KUKA KRL program: wkz6_an.src, wkz6_an.dat

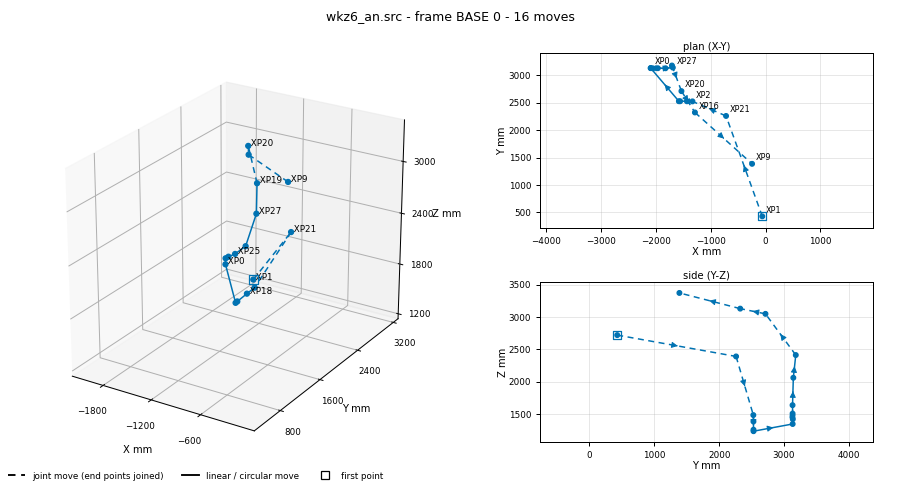
[picture p0: tool path of wkz6_an.src in frame BASE 0, 16 of 16 moves have a stored position in this frame; points joined in program order, loops and branches not executed]
--- wkz6_an.src ---
&ACCESS RVO4
&REL 71
&COMMENT Peg Grp AXOR
&PARAM DISKPATH = KRC:\R1\Program
&PARAM TEMPLATE = C:\KRC\Roboter\Template\vorgabe
&PARAM EDITMASK = *
DEF wkz6_an( )
;FOLD INI
  ;FOLD BASISTECH INI
    GLOBAL INTERRUPT DECL 3 WHEN $STOPMESS==TRUE DO IR_STOPM ( )
    INTERRUPT ON 3
    BAS (#INITMOV,0 )
  ;ENDFOLD (BASISTECH INI)
;FOLD GRIPPERTECH INI
USER_GRP(0,DUMMY,DUMMY,GDEFAULT)
;ENDFOLD (GRIPPERTECH INI)
  ;FOLD USER INI
    ;Make your modifications here

  ;ENDFOLD (USER INI)
;ENDFOLD (INI)

; Caracterização dos meios de produção
; Changes: Pega Gripper Axor/Atego
; Versão Atual:02/08/2015
; Name: P13.050-R3
; Docking

chk_w8_wechs_ok ( )     ; CHECK TOOL CHANGE

;FOLD PTP P1 CONT Vel=100 % PDAT1 Tool[6]:Gripper G0100R Base[0];%{PE}%R 8.2.20,%MKUKATPBASIS,%CMOVE,%VPTP,%P 1:PTP, 2:P1, 3:C_DIS, 5:100, 7:PDAT1
$BWDSTART=FALSE
PDAT_ACT=PPDAT1
FDAT_ACT=FP1
BAS(#PTP_PARAMS,100)
PTP XP1 C_DIS
;ENDFOLD

;FOLD WAIT FOR NOT ( IN 219 'Posicao p/ Acoplamento OK' ) CONT;%{PE}%R 8.2.20,%MKUKATPBASIS,%CEXT_WAIT_FOR,%VEXT_WAIT_FOR,%P 2:NOT, 4:, 5:$IN, 6:219, 7:Posicao p/ Acoplamento OK, 9:CONTINUE
CONTINUE
WAIT FOR  NOT ( $IN[219] )
;ENDFOLD
;FOLD WAIT FOR ( IN 201 'DOCK 6 Deposito Ocupado' ) CONT;%{PE}%R 8.2.20,%MKUKATPBASIS,%CEXT_WAIT_FOR,%VEXT_WAIT_FOR,%P 2:, 4:, 5:$IN, 6:201, 7:DOCK 6 Deposito Ocupado, 9:CONTINUE
CONTINUE
WAIT FOR  ( $IN[201] )
;ENDFOLD
;FOLD PULSE 207 'DOCK 6 Abrir Proteção' State=TRUE CONT Time=1 sec;%{PE}%R 8.2.20,%MKUKATPBASIS,%COUT,%VPULSE,%P 2:207, 3:DOCK 6 Abrir Proteção, 5:TRUE, 6:CONTINUE, 8:1
CONTINUE
PULSE($OUT[207], TRUE,1)
;ENDFOLD

;FOLD PTP P21 CONT Vel=100 % PDAT16 Tool[6]:Gripper G0100R Base[0];%{PE}%R 8.2.20,%MKUKATPBASIS,%CMOVE,%VPTP,%P 1:PTP, 2:P21, 3:C_DIS, 5:100, 7:PDAT16
$BWDSTART=FALSE
PDAT_ACT=PPDAT16
FDAT_ACT=FP21
BAS(#PTP_PARAMS,100)
PTP XP21 C_DIS
;ENDFOLD

;FOLD WAIT FOR ( IN 205 'DOCK 6 Proteção Aberta' ) CONT;%{PE}%R 8.2.20,%MKUKATPBASIS,%CEXT_WAIT_FOR,%VEXT_WAIT_FOR,%P 2:, 4:, 5:$IN, 6:205, 7:DOCK 6 Proteção Aberta, 9:CONTINUE
CONTINUE
WAIT FOR  ( $IN[205] )
;ENDFOLD
;FOLD WAIT FOR NOT ( IN 206 'DOCK 6 Proteção Fechada' ) CONT;%{PE}%R 8.2.20,%MKUKATPBASIS,%CEXT_WAIT_FOR,%VEXT_WAIT_FOR,%P 2:NOT, 4:, 5:$IN, 6:206, 7:DOCK 6 Proteção Fechada, 9:CONTINUE
CONTINUE
WAIT FOR  NOT ( $IN[206] )
;ENDFOLD

;FOLD PTP P2 CONT Vel=100 % PDAT7 Tool[6]:Gripper G0100R Base[0];%{PE}%R 8.2.20,%MKUKATPBASIS,%CMOVE,%VPTP,%P 1:PTP, 2:P2, 3:C_DIS, 5:100, 7:PDAT7
$BWDSTART=FALSE
PDAT_ACT=PPDAT7
FDAT_ACT=FP2
BAS(#PTP_PARAMS,100)
PTP XP2 C_DIS
;ENDFOLD
;FOLD LIN P18 CONT Vel=1 m/s CPDAT9 Tool[6]:Gripper G0100R Base[0];%{PE}%R 8.2.20,%MKUKATPBASIS,%CMOVE,%VLIN,%P 1:LIN, 2:P18, 3:C_DIS C_DIS, 5:1, 7:CPDAT9
$BWDSTART=FALSE
LDAT_ACT=LCPDAT9
FDAT_ACT=FP18
BAS(#CP_PARAMS,1)
LIN XP18 C_DIS C_DIS
;ENDFOLD
;FOLD LIN P22 CONT Vel=1 m/s CPDAT0 Tool[6]:Gripper G0100R Base[0];%{PE}%R 8.2.20,%MKUKATPBASIS,%CMOVE,%VLIN,%P 1:LIN, 2:P22, 3:C_DIS C_DIS, 5:1, 7:CPDAT0
$BWDSTART=FALSE
LDAT_ACT=LCPDAT0
FDAT_ACT=FP22
BAS(#CP_PARAMS,1)
LIN XP22 C_DIS C_DIS
;ENDFOLD

;FOLD WAIT FOR ( IN 222 'Liberacao p/ Desbloqueio' );%{PE}%R 8.2.20,%MKUKATPBASIS,%CEXT_WAIT_FOR,%VEXT_WAIT_FOR,%P 2:, 4:, 5:$IN, 6:222, 7:Liberacao p/ Desbloqueio, 9:
WAIT FOR  ( $IN[222] )
;ENDFOLD
;FOLD OUT 224 'Bloquear MPS' State=FALSE ;%{PE}%R 8.2.20,%MKUKATPBASIS,%COUT,%VOUTX,%P 2:224, 3:Bloquear MPS, 5:FALSE, 6:
$OUT[224]=FALSE
;ENDFOLD
;FOLD OUT 223 'Desbloquear MPS' State=TRUE ;%{PE}%R 8.2.20,%MKUKATPBASIS,%COUT,%VOUTX,%P 2:223, 3:Desbloquear MPS, 5:TRUE, 6:
$OUT[223]=TRUE
;ENDFOLD
;FOLD WAIT FOR ( IN 217 'MPS Destravado' );%{PE}%R 8.2.20,%MKUKATPBASIS,%CEXT_WAIT_FOR,%VEXT_WAIT_FOR,%P 2:, 4:, 5:$IN, 6:217, 7:MPS Destravado, 9:
WAIT FOR  ( $IN[217] )
;ENDFOLD
;FOLD WAIT FOR NOT ( IN 221 'MPS Travado' );%{PE}%R 8.2.20,%MKUKATPBASIS,%CEXT_WAIT_FOR,%VEXT_WAIT_FOR,%P 2:NOT, 4:, 5:$IN, 6:221, 7:MPS Travado, 9:
WAIT FOR  NOT ( $IN[221] )
;ENDFOLD

;FOLD ; POSICAO DE PEGA DO GRIPPER NO DOCKING;%{PE}%R 8.2.17,%MKUKATPBASIS,%CCOMMENT,%VNORMAL,%P 2:POSICAO DE PEGA DO GRIPPER NO DOCKING
;ENDFOLD
;FOLD LIN P4 Vel=0.2 m/s CPDAT16 Tool[8]:Tool Changer Base[0];%{PE}%R 8.2.20,%MKUKATPBASIS,%CMOVE,%VLIN,%P 1:LIN, 2:P4, 3:, 5:0.2, 7:CPDAT16
$BWDSTART=FALSE
LDAT_ACT=LCPDAT16
FDAT_ACT=FP4
BAS(#CP_PARAMS,0.2)
LIN XP4
;ENDFOLD

;FOLD WAIT FOR ( IN 219 'Posicao p/ Acoplamento OK' );%{PE}%R 8.2.20,%MKUKATPBASIS,%CEXT_WAIT_FOR,%VEXT_WAIT_FOR,%P 2:, 4:, 5:$IN, 6:219, 7:Posicao p/ Acoplamento OK, 9:
WAIT FOR  ( $IN[219] )
;ENDFOLD
;FOLD WAIT Time=0.5 sec;%{PE}%R 8.2.20,%MKUKATPBASIS,%CWAIT,%VWAIT,%P 3:0.5
WAIT SEC 0.5
;ENDFOLD
;FOLD OUT 223 'Desbloquear MPS' State=FALSE ;%{PE}%R 8.2.20,%MKUKATPBASIS,%COUT,%VOUTX,%P 2:223, 3:Desbloquear MPS, 5:FALSE, 6:
$OUT[223]=FALSE
;ENDFOLD
;FOLD OUT 224 'Bloquear MPS' State=TRUE ;%{PE}%R 8.2.20,%MKUKATPBASIS,%COUT,%VOUTX,%P 2:224, 3:Bloquear MPS, 5:TRUE, 6:
$OUT[224]=TRUE
;ENDFOLD
;FOLD WAIT FOR NOT ( IN 217 'MPS Destravado' );%{PE}%R 8.2.20,%MKUKATPBASIS,%CEXT_WAIT_FOR,%VEXT_WAIT_FOR,%P 2:NOT, 4:, 5:$IN, 6:217, 7:MPS Destravado, 9:
WAIT FOR  NOT ( $IN[217] )
;ENDFOLD
;FOLD WAIT FOR ( IN 221 'MPS Travado' );%{PE}%R 8.2.20,%MKUKATPBASIS,%CEXT_WAIT_FOR,%VEXT_WAIT_FOR,%P 2:, 4:, 5:$IN, 6:221, 7:MPS Travado, 9:
WAIT FOR  ( $IN[221] )
;ENDFOLD
;FOLD IBUS ON SEGMENT_4;%{PE}%R 8.2.20,%MKUKATPBASIS,%CIBUS,%VMAP,%P 2:#ON, 3:4
$IBUS_ON=IBUS_SEGMENT[4]
$IBUS_OFF=0
;ENDFOLD
;FOLD WAIT Time=0.5 sec;%{PE}%R 8.2.20,%MKUKATPBASIS,%CWAIT,%VWAIT,%P 3:0.5
WAIT SEC 0.5
;ENDFOLD

; Verifica Grampos da Garra Fechados
chk_w6_grp3_clo()
chk_w6_grp4_clo()
chk_w6_grp5_clo()
chk_w6_grp6_clo()
chk_w6_grp7_clo()

;FOLD LIN P0 CONT Vel=0.3 m/s CPDAT1 Tool[6]:Gripper G0100R Base[0];%{PE}%R 8.2.20,%MKUKATPBASIS,%CMOVE,%VLIN,%P 1:LIN, 2:P0, 3:C_DIS C_DIS, 5:0.3, 7:CPDAT1
$BWDSTART=FALSE
LDAT_ACT=LCPDAT1
FDAT_ACT=FP0
BAS(#CP_PARAMS,0.3)
LIN XP0 C_DIS C_DIS
;ENDFOLD
;FOLD LIN P12 CONT Vel=0.5 m/s CPDAT7 Tool[6]:Gripper G0100R Base[0];%{PE}%R 8.2.20,%MKUKATPBASIS,%CMOVE,%VLIN,%P 1:LIN, 2:P12, 3:C_DIS C_DIS, 5:0.5, 7:CPDAT7
$BWDSTART=FALSE
LDAT_ACT=LCPDAT7
FDAT_ACT=FP12
BAS(#CP_PARAMS,0.5)
LIN XP12 C_DIS C_DIS
;ENDFOLD

;FOLD WAIT FOR NOT ( IN 201 'DOCK 6 Deposito Ocupado' ) CONT;%{PE}%R 8.2.20,%MKUKATPBASIS,%CEXT_WAIT_FOR,%VEXT_WAIT_FOR,%P 2:NOT, 4:, 5:$IN, 6:201, 7:DOCK 6 Deposito Ocupado, 9:CONTINUE
CONTINUE
WAIT FOR  NOT ( $IN[201] )
;ENDFOLD
;FOLD WAIT FOR ( IN 219 'Posicao p/ Acoplamento OK' ) CONT;%{PE}%R 8.2.20,%MKUKATPBASIS,%CEXT_WAIT_FOR,%VEXT_WAIT_FOR,%P 2:, 4:, 5:$IN, 6:219, 7:Posicao p/ Acoplamento OK, 9:CONTINUE
CONTINUE
WAIT FOR  ( $IN[219] )
;ENDFOLD

;FOLD LIN P24 CONT Vel=1 m/s CPDAT11 Tool[6]:Gripper G0100R Base[0];%{PE}%R 8.2.20,%MKUKATPBASIS,%CMOVE,%VLIN,%P 1:LIN, 2:P24, 3:C_DIS C_DIS, 5:1, 7:CPDAT11
$BWDSTART=FALSE
LDAT_ACT=LCPDAT11
FDAT_ACT=FP24
BAS(#CP_PARAMS,1)
LIN XP24 C_DIS C_DIS
;ENDFOLD
;FOLD LIN P25 CONT Vel=1 m/s CPDAT17 Tool[6]:Gripper G0100R Base[0];%{PE}%R 8.2.20,%MKUKATPBASIS,%CMOVE,%VLIN,%P 1:LIN, 2:P25, 3:C_DIS C_DIS, 5:1, 7:CPDAT17
$BWDSTART=FALSE
LDAT_ACT=LCPDAT17
FDAT_ACT=FP25
BAS(#CP_PARAMS,1)
LIN XP25 C_DIS C_DIS
;ENDFOLD
;FOLD LIN P26 CONT Vel=1 m/s CPDAT18 Tool[6]:Gripper G0100R Base[0];%{PE}%R 8.2.20,%MKUKATPBASIS,%CMOVE,%VLIN,%P 1:LIN, 2:P26, 3:C_DIS C_DIS, 5:1, 7:CPDAT18
$BWDSTART=FALSE
LDAT_ACT=LCPDAT18
FDAT_ACT=FP26
BAS(#CP_PARAMS,1)
LIN XP26 C_DIS C_DIS
;ENDFOLD
;FOLD LIN P27 CONT Vel=2 m/s CPDAT19 Tool[6]:Gripper G0100R Base[0];%{PE}%R 8.2.20,%MKUKATPBASIS,%CMOVE,%VLIN,%P 1:LIN, 2:P27, 3:C_DIS C_DIS, 5:2, 7:CPDAT19
$BWDSTART=FALSE
LDAT_ACT=LCPDAT19
FDAT_ACT=FP27
BAS(#CP_PARAMS,2)
LIN XP27 C_DIS C_DIS
;ENDFOLD
;FOLD LIN P19 CONT Vel=2 m/s CPDAT15 Tool[6]:Gripper G0100R Base[0];%{PE}%R 8.2.20,%MKUKATPBASIS,%CMOVE,%VLIN,%P 1:LIN, 2:P19, 3:C_DIS C_DIS, 5:2, 7:CPDAT15
$BWDSTART=FALSE
LDAT_ACT=LCPDAT15
FDAT_ACT=FP19
BAS(#CP_PARAMS,2)
LIN XP19 C_DIS C_DIS
;ENDFOLD
;FOLD PTP P20 CONT Vel=100 % PDAT15 Tool[6]:Gripper G0100R Base[0];%{PE}%R 8.2.20,%MKUKATPBASIS,%CMOVE,%VPTP,%P 1:PTP, 2:P20, 3:C_DIS, 5:100, 7:PDAT15
$BWDSTART=FALSE
PDAT_ACT=PPDAT15
FDAT_ACT=FP20
BAS(#PTP_PARAMS,100)
PTP XP20 C_DIS
;ENDFOLD
;FOLD PTP P16 CONT Vel=100 % PDAT12 Tool[6]:Gripper G0100R Base[0];%{PE}%R 8.2.20,%MKUKATPBASIS,%CMOVE,%VPTP,%P 1:PTP, 2:P16, 3:C_DIS, 5:100, 7:PDAT12
$BWDSTART=FALSE
PDAT_ACT=PPDAT12
FDAT_ACT=FP16
BAS(#PTP_PARAMS,100)
PTP XP16 C_DIS
;ENDFOLD
;FOLD PTP P9 CONT Vel=100 % PDAT4 Tool[6]:Gripper G0100R Base[0];%{PE}%R 8.2.20,%MKUKATPBASIS,%CMOVE,%VPTP,%P 1:PTP, 2:P9, 3:C_DIS, 5:100, 7:PDAT4
$BWDSTART=FALSE
PDAT_ACT=PPDAT4
FDAT_ACT=FP9
BAS(#PTP_PARAMS,100)
PTP XP9 C_DIS
;ENDFOLD

END

--- wkz6_an.dat ---
&ACCESS RVO4
&REL 71
&COMMENT Peg Grp AXOR
&PARAM DISKPATH = KRC:\R1\Program
&PARAM TEMPLATE = C:\KRC\Roboter\Template\vorgabe
&PARAM EDITMASK = *
DEFDAT  wkz6_an
;FOLD EXTERNAL DECLARATIONS;%{PE}%MKUKATPBASIS,%CEXT,%VCOMMON,%P
;FOLD GRIPPERTECH EXT
EXT  H50 (INT  :IN,INT  :IN,INT  :IN,GRP_TYP  :IN )
;ENDFOLD (GRIPPERTECH EXT)
;FOLD SPOTTECH EXT
EXT  USERSPOT (S_COMMAND  :IN,SPOT_TYPE  :IN )
;ENDFOLD (SPOTTECH EXT)
;FOLD BASISTECH EXT;%{PE}%MKUKATPBASIS,%CEXT,%VEXT,%P
EXT  BAS (BAS_COMMAND  :IN,REAL  :IN )
DECL INT SUCCESS
;ENDFOLD (BASISTECH EXT)
;FOLD USER EXT;%{E}%MKUKATPUSER,%CEXT,%VEXT,%P
;Make your modifications here

;ENDFOLD (USER EXT)
;ENDFOLD (EXTERNAL DECLARATIONS)
DECL BASIS_SUGG_T LAST_BASIS={POINT1[] "P0                      ",POINT2[] "P0                      ",CP_PARAMS[] "CPDAT0                  ",PTP_PARAMS[] "PDAT0                   ",CONT[] "                        ",CP_VEL[] "0.2                     ",PTP_VEL[] "100                     ",SYNC_PARAMS[] "SYNCDAT                 ",SPL_NAME[] "S0                      "}
DECL E6POS XP2={X -1334.70801,Y 2526.76001,Z 1488.44397,A -20.9060402,B 43.2974091,C 166.070602,S 2,T 10,E1 -276.315094,E2 0.0,E3 0.0,E4 0.0,E5 0.0,E6 0.0}
DECL FDAT FP2={TOOL_NO 8,BASE_NO 0,IPO_FRAME #BASE,POINT2[] " ",TQ_STATE FALSE}
DECL E6POS XP4={X -1582.73999,Y 2529.76489,Z 1240.026,A -20.81633,B 42.8571701,C 165.799393,S 2,T 10,E1 -276.288391,E2 0.0,E3 0.0,E4 0.0,E5 0.0,E6 0.0}
DECL FDAT FP4={TOOL_NO 8,BASE_NO 0,IPO_FRAME #BASE,POINT2[] " ",TQ_STATE FALSE}
DECL E6POS XP9={X -246.532501,Y 1387.03601,Z 3371.896,A -169.795593,B 6.91202211,C 129.772507,S 2,T 34,E1 -430.979797,E2 0.0,E3 0.0,E4 0.0,E5 0.0,E6 0.0}
DECL FDAT FP9={TOOL_NO 6,BASE_NO 0,IPO_FRAME #BASE,POINT2[] " ",TQ_STATE FALSE}
DECL PDAT PPDAT4={VEL 100.0,ACC 100.0,APO_DIST 0.0,APO_MODE #CDIS}
DECL E6POS XP12={X -2096.30688,Y 3135.69604,Z 1425.60205,A -0.0780687928,B 45.1058998,C -104.320198,S 2,T 10,E1 -276.26181,E2 0.0,E3 0.0,E4 0.0,E5 0.0,E6 0.0}
DECL FDAT FP12={TOOL_NO 6,BASE_NO 0,IPO_FRAME #BASE,POINT2[] " ",TQ_STATE FALSE}
DECL LDAT LCPDAT7={VEL 2.0,ACC 100.0,APO_DIST 20.0,APO_FAC 50.0,AXIS_VEL 100.0,AXIS_ACC 100.0,ORI_TYP #VAR,CIRC_TYP #BASE,JERK_FAC 50.0,GEAR_JERK 50.0,EXAX_IGN 0}
DECL PDAT PPDAT7={VEL 100.0,ACC 100.0,APO_DIST 50.0,APO_MODE #CDIS}
DECL E6POS XP16={X -1289.547,Y 2324.76294,Z 3130.05688,A -36.2241287,B 48.9362907,C -95.0278778,S 2,T 34,E1 -331.860504,E2 0.0,E3 0.0,E4 0.0,E5 0.0,E6 0.0}
DECL FDAT FP16={TOOL_NO 6,BASE_NO 0,IPO_FRAME #BASE,POINT2[] " ",TQ_STATE FALSE}
DECL PDAT PPDAT12={VEL 100.0,ACC 100.0,APO_DIST 100.0,APO_MODE #CDIS}
DECL E6POS XP18={X -1434.875,Y 2528.70508,Z 1389.41895,A -20.3609009,B 42.94133,C 166.110596,S 2,T 10,E1 -276.315002,E2 0.0,E3 0.0,E4 0.0,E5 0.0,E6 0.0}
DECL FDAT FP18={TOOL_NO 8,BASE_NO 0,IPO_FRAME #BASE,POINT2[] " ",TQ_STATE FALSE}
DECL LDAT LCPDAT9={VEL 2.0,ACC 100.0,APO_DIST 10.0,APO_FAC 50.0,AXIS_VEL 100.0,AXIS_ACC 100.0,ORI_TYP #VAR,CIRC_TYP #BASE,JERK_FAC 50.0,GEAR_JERK 50.0,EXAX_IGN 0}
DECL E6POS XP19={X -1709.26904,Y 3181.41309,Z 2414.36304,A 0.598406494,B 55.2073517,C -102.179604,S 2,T 10,E1 -276.258514,E2 0.0,E3 0.0,E4 0.0,E5 0.0,E6 0.0}
DECL FDAT FP19={TOOL_NO 6,BASE_NO 0,IPO_FRAME #BASE,POINT2[] " ",TQ_STATE FALSE}
DECL E6POS XP20={X -1535.84998,Y 2714.00806,Z 3049.51196,A 15.8610601,B 57.4065895,C -83.8867493,S 2,T 10,E1 -276.258606,E2 0.0,E3 0.0,E4 0.0,E5 0.0,E6 0.0}
DECL FDAT FP20={TOOL_NO 6,BASE_NO 0,IPO_FRAME #BASE,POINT2[] " ",TQ_STATE FALSE}
DECL PDAT PPDAT15={VEL 100.0,ACC 100.0,APO_DIST 100.0,APO_MODE #CDIS}
DECL GRP_SUGG_T LAST_GRP={NUMBER[] "14                      ",STATE[] "2                       ",PARAMS[] "GDAT5                   "}
DECL GRP_TYP GGDAT14={G_APO #NO,GRP_TIME 0.200000003,CTRL #OFF,DLY 0,DST 1}
DECL GRP_TYP GGDAT15={G_APO #NO,GRP_TIME 0.200000003,CTRL #OFF,DLY 0,DST 1}
DECL GRP_TYP GGDAT16={G_APO #NO,GRP_TIME 0.200000003,CTRL #OFF,DLY 0,DST 1}
DECL GRP_TYP GGDAT17={G_APO #NO,GRP_TIME 0.200000003,CTRL #OFF,DLY 0,DST 1}
DECL GRP_TYP GGDAT18={G_APO #NO,GRP_TIME 0.200000003,CTRL #OFF,DLY 0,DST 1}
DECL GRP_TYP GGDAT19={G_APO #NO,GRP_TIME 0.200000003,CTRL #OFF,DLY 0,DST 1}
DECL E6POS XP21={X -721.451416,Y 2260.86401,Z 2392.80103,A -69.6591873,B 42.6547394,C -179.8293,S 2,T 10,E1 -276.320099,E2 0.0,E3 0.0,E4 0.0,E5 0.0,E6 0.0}
DECL FDAT FP21={TOOL_NO 8,BASE_NO 0,IPO_FRAME #BASE,POINT2[] " ",TQ_STATE FALSE}
DECL PDAT PPDAT16={VEL 100.0,ACC 100.0,APO_DIST 100.0,APO_MODE #CDIS}
DECL LDAT LCPDAT0={VEL 2.0,ACC 100.0,APO_DIST 10.0,APO_FAC 50.0,AXIS_VEL 100.0,AXIS_ACC 100.0,ORI_TYP #VAR,CIRC_TYP #BASE,JERK_FAC 50.0,GEAR_JERK 50.0,EXAX_IGN 0}
DECL E6POS XP22={X -1560.15796,Y 2529.604,Z 1262.86804,A -20.8148899,B 42.858139,C 165.801605,S 2,T 10,E1 -276.314697,E2 0.0,E3 0.0,E4 0.0,E5 0.0,E6 0.0}
DECL FDAT FP22={TOOL_NO 8,BASE_NO 0,IPO_FRAME #BASE,POINT2[] " ",TQ_STATE FALSE}
DECL LDAT LCPDAT11={VEL 2.0,ACC 100.0,APO_DIST 20.0,APO_FAC 50.0,AXIS_VEL 100.0,AXIS_ACC 100.0,ORI_TYP #VAR,CIRC_TYP #BASE,JERK_FAC 50.0,GEAR_JERK 50.0,EXAX_IGN 0}
DECL E6POS XP24={X -2053.76294,Y 3129.93408,Z 1457.85706,A 0.313883901,B 46.6480103,C -104.005699,S 2,T 10,E1 -276.260712,E2 0.0,E3 0.0,E4 0.0,E5 0.0,E6 0.0}
DECL FDAT FP24={TOOL_NO 6,BASE_NO 0,IPO_FRAME #BASE,POINT2[] " ",TQ_STATE FALSE}
DECL E6POS XP25={X -1966.83496,Y 3132.13403,Z 1511.82605,A 0.0466624014,B 49.53125,C -104.139999,S 2,T 10,E1 -276.258606,E2 0.0,E3 0.0,E4 0.0,E5 0.0,E6 0.0}
DECL FDAT FP25={TOOL_NO 6,BASE_NO 0,IPO_FRAME #BASE,POINT2[] " ",TQ_STATE FALSE}
DECL E6POS XP26={X -1826.46497,Y 3131.44409,Z 1641.16504,A 0.067385383,B 50.164299,C -103.951599,S 2,T 10,E1 -276.258789,E2 0.0,E3 0.0,E4 0.0,E5 0.0,E6 0.0}
DECL FDAT FP26={TOOL_NO 6,BASE_NO 0,IPO_FRAME #BASE,POINT2[] " ",TQ_STATE FALSE}
DECL E6POS XP27={X -1693.302,Y 3143.63599,Z 2063.99707,A 0.53788811,B 54.4673309,C -102.427696,S 2,T 10,E1 -276.258606,E2 0.0,E3 0.0,E4 0.0,E5 0.0,E6 0.0}
DECL FDAT FP27={TOOL_NO 6,BASE_NO 0,IPO_FRAME #BASE,POINT2[] " ",TQ_STATE FALSE}
DECL LDAT LCPDAT15={VEL 2.0,ACC 100.0,APO_DIST 50.0,APO_FAC 50.0,AXIS_VEL 100.0,AXIS_ACC 100.0,ORI_TYP #VAR,CIRC_TYP #BASE,JERK_FAC 50.0,GEAR_JERK 50.0,EXAX_IGN 0}
DECL LDAT LCPDAT16={VEL 2.0,ACC 100.0,APO_DIST 100.0,APO_FAC 50.0,AXIS_VEL 100.0,AXIS_ACC 100.0,ORI_TYP #VAR,CIRC_TYP #BASE,JERK_FAC 50.0,GEAR_JERK 50.0,EXAX_IGN 0}
DECL LDAT LCPDAT17={VEL 2.0,ACC 100.0,APO_DIST 20.0,APO_FAC 50.0,AXIS_VEL 100.0,AXIS_ACC 100.0,ORI_TYP #VAR,CIRC_TYP #BASE,JERK_FAC 50.0,GEAR_JERK 50.0,EXAX_IGN 0}
DECL LDAT LCPDAT18={VEL 2.0,ACC 100.0,APO_DIST 20.0,APO_FAC 50.0,AXIS_VEL 100.0,AXIS_ACC 100.0,ORI_TYP #VAR,CIRC_TYP #BASE,JERK_FAC 50.0,GEAR_JERK 50.0,EXAX_IGN 0}
DECL LDAT LCPDAT19={VEL 2.0,ACC 100.0,APO_DIST 50.0,APO_FAC 50.0,AXIS_VEL 100.0,AXIS_ACC 100.0,ORI_TYP #VAR,CIRC_TYP #BASE,JERK_FAC 50.0,GEAR_JERK 50.0,EXAX_IGN 0}
DECL GRP_TYP GGDAT1={G_APO #NO,GRP_TIME 0.200000003,CTRL #OFF,DLY 0,DST 1}
DECL GRP_TYP GGDAT2={G_APO #NO,GRP_TIME 0.200000003,CTRL #OFF,DLY 0,DST 1}
DECL GRP_TYP GGDAT3={G_APO #NO,GRP_TIME 0.200000003,CTRL #OFF,DLY 0,DST 1}
DECL GRP_TYP GGDAT4={G_APO #NO,GRP_TIME 0.200000003,CTRL #OFF,DLY 0,DST 1}
DECL GRP_TYP GGDAT5={G_APO #NO,GRP_TIME 0.200000003,CTRL #OFF,DLY 0,DST 1}
DECL GRP_TYP GGDAT6={G_APO #NO,GRP_TIME 0.200000003,CTRL #OFF,DLY 0,DST 1}
DECL GRP_TYP GCONT={G_APO #YES,GRP_TIME 0.0,CTRL #OFF,DLY 0,DST 0}
DECL E6POS XP1={X -60.1240082,Y 428.122406,Z 2721.90894,A 9.3139267,B -8.93749809,C -139.628693,S 2,T 2,E1 1119.99695,E2 0.0,E3 0.0,E4 0.0,E5 0.0,E6 0.0}
DECL FDAT FP1={TOOL_NO 8,BASE_NO 0,IPO_FRAME #BASE,POINT2[] " ",TQ_STATE FALSE}
DECL PDAT PPDAT1={VEL 100.0,ACC 100.0,APO_DIST 100.0,APO_MODE #CDIS}
DECL LDAT LCPDAT1={VEL 2.0,ACC 100.0,APO_DIST 10.0,APO_FAC 50.0,AXIS_VEL 100.0,AXIS_ACC 100.0,ORI_TYP #VAR,CIRC_TYP #BASE,JERK_FAC 50.0,GEAR_JERK 50.0,EXAX_IGN 0}
DECL E6POS XP0={X -2096.63696,Y 3133.30103,Z 1351.18201,A -0.122571997,B 44.8263588,C -104.667297,S 2,T 10,E1 -276.299286,E2 0.0,E3 0.0,E4 0.0,E5 0.0,E6 0.0}
DECL FDAT FP0={TOOL_NO 6,BASE_NO 0,IPO_FRAME #BASE,POINT2[] " ",TQ_STATE FALSE}
ENDDAT
